FUNCTION_BLOCK fbLoadCell
VAR
	wStatus		AT %I* : WORD;	// .1-Overrange, .3-Data invalid, .6-Error, .7-Calib in progress, .9-Steady state, .13-SyncErr, .15-TxPDO_Toggle
	rValue		AT %I* : REAL;	// Wartość siły w [N]
	wControl	AT %Q* : WORD;	// .0-Start calibration, .1-Disable calib., .2-InputFreeze, .4-Tara                  
END_VAR

PROPERTY propDisableCalibration : BOOL
GET
propDisableCalibration:= wControl.1;
END_GET
SET
wControl.1 := propDisableCalibration;
END_SET
END_PROPERTY

PROPERTY propIsCalibrationInProgress : BOOL
GET
propIsCalibrationInProgress := wStatus.7;
END_GET
END_PROPERTY

PROPERTY propIsValueReady : BOOL
GET
propIsValueReady := NOT wStatus.1 AND NOT wStatus.3 AND NOT wStatus.6 AND NOT wStatus.7 AND NOT wStatus.13;
END_GET
END_PROPERTY

PROPERTY propStartCalibration : BOOL
GET
propStartCalibration:= wControl.0;
END_GET
SET
wControl.0 := propStartCalibration;
END_SET
END_PROPERTY

PROPERTY propValue : REAL
GET
propValue := rValue;
END_GET
END_PROPERTY

END_FUNCTION_BLOCK

(* stored: Version 1.1.0.1, ProductVersion 3.1.4024.12
   POU fbLoadCell: Id {4ed80c1b-acfa-4f29-a893-2740788a7820}, SpecialFunc None
   Property propDisableCalibration: Id {7077f5d9-6359-47e8-9d1a-003d37246b4a}
   Get Get: Id {c6f0b1cc-f3d0-4af3-b05e-e883918721d3}
   Set Set: Id {28f9980e-c46e-4651-b4ab-96f485fdecfd}
   Property propIsCalibrationInProgress: Id {85dd532d-ef43-44ed-955f-aa51b217b6ec}
   Get Get: Id {1cf7078d-bb0f-4041-b1a6-2cf1203bafab}
   Property propIsValueReady: Id {64a10cc6-17ca-42d7-9b2c-6a03f9792cc6}
   Get Get: Id {b8e8d96a-e207-49d4-af55-1c4f805642cd}
   Property propStartCalibration: Id {b258b86e-fe2b-4f79-a73b-702e70425705}
   Get Get: Id {9fa0dfa0-6b93-4e1d-b41a-40bb28a04bc1}
   Set Set: Id {0c004399-18c6-43a3-8cb6-9249359a6ed0}
   Property propValue: Id {76bfce06-1cae-4b0a-a168-019ea64560d0}
   Get Get: Id {0e89c5a7-702d-46f5-b52c-284658db08c2} *)
